# EPICS autosave request: iocBoot/iocScanLib/auto_settings.req
file "scanLib.req", P=$(P), R=$(R)
file "scanLib_settings.req", P=$(P), R=$(R)
